ABB RobotStudio station: Sesion7_Parte1_interrupciones.rsstn

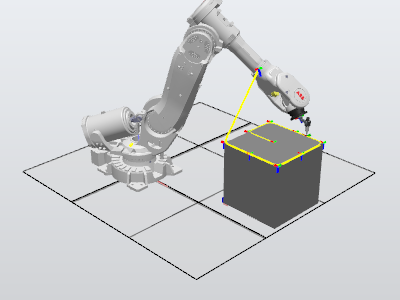
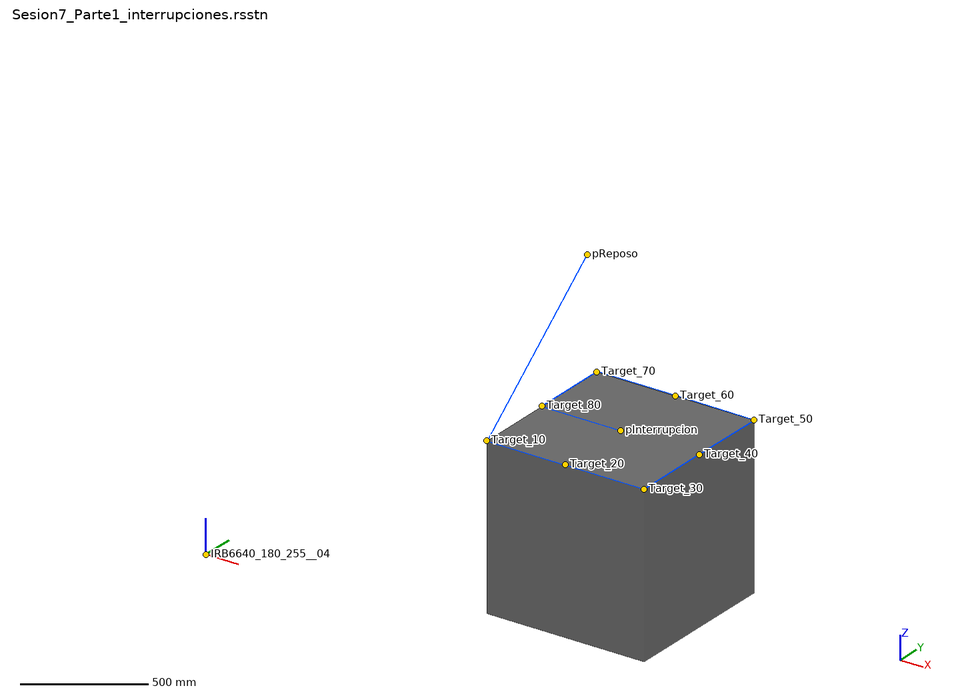
[picture v1: parts stored in the station drawn from their meshes, with robot base, taught points and paths (robot models come from the ABB library and are not in the file)]
Station borr (saved by RobotStudio 24.1.10713.1)
Controller Controlador10
  mechanical unit ROB_1: IRB6640_180_255__04, 6 joints, base frame (0, 0, 0) mm
Layout (positions relative to the parent item):
  - IRB6640_180_255__04 [mechanism, from %ABB.RobotStudio.Models.IRB6640%\IRB6640_180_255_G_04.rslib] at (0, 0, 0) mm; joint values [0.569, 0.4564, 0.2981, -0.9875, 0.4087, 1.4142] (rad or m)
  - MyTool [mechanism, from Training Objects\myTool.rslib] at (1608.5, 950, 950.53) mm, rotated rx -180 ry 38 rz 180 deg
  - Pieza_1 [part], size 750 x 750 x 750 mm
Attachment: MyTool is attached to IRB6640_180_255__04 / Link6
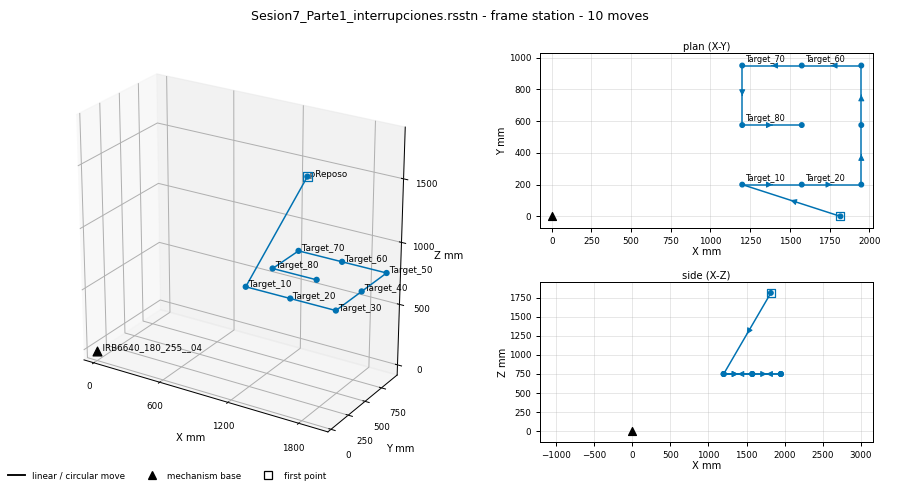
[picture p0: tool path of Sesion7_Parte1_interrupciones.rsstn in frame station, 10 of 10 moves have a stored position in this frame; points joined in program order, loops and branches not executed]
Targets, tools, work objects and paths stored in the station, written as RAPID:
! task T_ROB1
MODULE CalibData
  PERS tooldata MyTool:=[TRUE,[[31.792631019,0,229.638935148],[0.945518576,0,0.325568154,0]],[1,[0,0,1],[1,0,0,0],0,0,0]];
  TASK PERS wobjdata Workobject_1:=[FALSE,TRUE,"",[[1200,200,0],[1,0,0,0]],[[0,0,0],[1,0,0,0]]];
ENDMODULE

! task T_ROB1
MODULE Module1
  CONST robtarget Target_10:=[[0,0,750],[0,0,1,0],[0,-1,0,0],[9E+09,9E+09,9E+09,9E+09,9E+09,9E+09]];
  CONST robtarget Target_20:=[[375,0,750],[0,0,1,0],[0,-1,0,0],[9E+09,9E+09,9E+09,9E+09,9E+09,9E+09]];
  CONST robtarget Target_30:=[[750,0,750],[0,0,1,0],[0,-1,0,0],[9E+09,9E+09,9E+09,9E+09,9E+09,9E+09]];
  CONST robtarget Target_40:=[[750,375,750],[0,0,1,0],[0,-1,0,0],[9E+09,9E+09,9E+09,9E+09,9E+09,9E+09]];
  CONST robtarget Target_50:=[[750,750,750],[0,0,1,0],[0,-1,0,0],[9E+09,9E+09,9E+09,9E+09,9E+09,9E+09]];
  CONST robtarget Target_60:=[[375,750,750],[0,0,1,0],[0,-1,0,0],[9E+09,9E+09,9E+09,9E+09,9E+09,9E+09]];
  CONST robtarget Target_70:=[[0,750,750],[0,0,1,0],[0,0,0,0],[9E+09,9E+09,9E+09,9E+09,9E+09,9E+09]];
  CONST robtarget Target_80:=[[0,375,750],[0,0,1,0],[0,0,0,0],[9E+09,9E+09,9E+09,9E+09,9E+09,9E+09]];
  CONST robtarget pInterrupcion:=[[375,375,750],[0,0,1,0],[0,0,0,0],[9E+09,9E+09,9E+09,9E+09,9E+09,9E+09]];
  CONST robtarget pReposo:=[[1818.681916784,0,1812.64730631],[0.190808996,0,0.981627183,0],[0,0,0,0],[9E+09,9E+09,9E+09,9E+09,9E+09,9E+09]];
  PROC Path_10()
    MoveL pReposo,v1000,z100,MyTool\WObj:=wobj0;
    MoveL Target_10,v1000,z100,MyTool\WObj:=Workobject_1;
    MoveL Target_20,v1000,z100,MyTool\WObj:=Workobject_1;
    MoveL Target_30,v1000,z100,MyTool\WObj:=Workobject_1;
    MoveL Target_40,v1000,z100,MyTool\WObj:=Workobject_1;
    MoveL Target_50,v1000,z100,MyTool\WObj:=Workobject_1;
    MoveL Target_60,v1000,z100,MyTool\WObj:=Workobject_1;
    MoveL Target_70,v1000,z100,MyTool\WObj:=Workobject_1;
    MoveL Target_80,v1000,z100,MyTool\WObj:=Workobject_1;
    MoveL pInterrupcion,v1000,z100,MyTool\WObj:=Workobject_1;
  ENDPROC
ENDMODULE

